	3: (* === Wait & process MB response *)
		IF NOT MB_Start THEN
			IF MB_MASTER.MB_Error=0 THEN
				CASE VARS[VarCnt].FunCode OF
					1,2,3,4:
						IF VARS[VarCnt].Variable_Size=200 THEN
							COPY_32SWAP16(ADR(MB_Resp.Data), VARS[VarCnt].Variable);
						ELSIF VARS[VarCnt].Variable_Size>1 THEN
							MEMCPY(ADR(MB_Resp.Data), VARS[VarCnt].Variable, 2*VARS[VarCnt].Variable_Size);
						ELSE
							VARS[VarCnt].Variable^:=MB_Resp.Data[0];
						END_IF
				END_CASE
				MB_Lock:=FALSE;
				(* Signal error recovery *)
				IF VARS_Alarm=TRUE AND VarCnt=VarAlarm THEN
					LogEv(EL_Wrn,EO_MODBUS,ID,5,'');
					VARS_Alarm:=FALSE;
				END_IF
				(* Next var *)
				VarCnt:=VarCnt+1;
				VarSta:=2;
			ELSE
				IF VarRetry<3 THEN
					VarRetry:=VarRetry+1;
					MB_Start:=TRUE;
				ELSE
					MB_Lock:=FALSE;
					(* Signal error *)
					IF VARS_Alarm=FALSE THEN
						LogEv(EL_Wrn,EO_MODBUS,ID,3,INT_TO_STRING(MB_MASTER.MB_Error));
						VARS_Alarm:=TRUE;
						VarAlarm:=VarCnt-1;
					END_IF
					(* Next var *)
					VarCnt:=VarCnt+1;
					VarSta:=2;
				END_IF
			END_IF
		END_IF

ELSE
	VarSta:=0;
END_CASE*)
;
END_ACTION

(* POU Plant_Objects/obj_MODBUS_TCP, ST *)
FUNCTION_BLOCK obj_MODBUS_TCP
(* === MODBUS-TCP PROTOCOL INTERFACE ===
   v1.0[10/06/15] - Create
*)
VAR CONSTANT
	VARS_Max	: BYTE := 32;
END_VAR
VAR_INPUT
	(* Settings *)
	ID			: BYTE;
	IP			: STRING;
	PORT		: WORD:=502;
	(* Interface *)
	MB_MASTER	: ETHERNET_MODBUSMASTER_TCP;
	MB_READBUF	: ARRAY [0..128] OF WORD;
	MB_WRITEBUF : ARRAY [0..128] OF WORD;
	MB_Start	: BOOL;
	MB_Lock		: BOOL;
	(* Variables management *)
	VARS_En		: BOOL;
	VARS		: ARRAY [0..VARS_Max] OF typ_MODBUS_VAR;
	VARS_Check	: BOOL;
	VARS_Alarm	: BOOL;
	(* Variables allocation *)
	VAR_Pointer : POINTER TO ARRAY[0..99] OF WORD;
	VAR_Cfg		: POINTER TO typ_MODBUS_VAR;
END_VAR
VAR_OUTPUT
	(* Status *)
	Status_Log	: BYTE;
	Status_Vis	: DWORD;
END_VAR
VAR
	sta         : BYTE :=0;
	i			: BYTE;
	j			: BYTE;
	Alarm		: FLT_EVENT;

	VarTmr		: TON := (PT:=T#1s);
	VarSta		: BYTE; (* Status *)
	VarCnt		: BYTE; (* Scan counter *)
	VarRetry	: BYTE;
	VarAlarm	: BYTE; (* Last variable with errors *)
END_VAR
MB_MASTER( strIP_ADDRESS:=IP, wPORT:=PORT, tTIME_OUT:=T#1s, (*xCONNECT:=TRUE,*)
		   ptREAD_DATA:=ADR(MB_READBUF), ptSEND_DATA:=ADR(MB_WRITEBUF), xSEND:=MB_Start );

IF sta=0 THEN
	MB_MASTER.xCONNECT:=TRUE;
	sta:=1;
END_IF

(* Process variable management *)
IF VARS_En THEN VARS_Process(); END_IF

(* Check status *)
Alarm(IN:=(MB_MASTER.wERROR<>0));
IF Alarm.EVH THEN
	(*LogEv(SEL(MB_MASTER.wERROR>0,EL_Wrn,EL_Alarm),EO_MODBUS_TCP,ID,1,WORD_TO_STRING(MB_MASTER.wERROR));*)
	(*LogEv(EL_Alarm,EO_MODBUS_TCP,ID,1,WORD_TO_STRING(MB_MASTER.wERROR));*);
END_IF
IF Alarm.EVL THEN
	(*LogEv(EL_Log,EO_MODBUS_TCP,ID,2,'');*);
END_IF

(* Log/visu status *)
   IF Alarm.IN   THEN Status_Log:=2; Status_Vis:=COLOR_RED;
ELSIF Vars_Alarm THEN Status_Log:=1; Status_Vis:=COLOR_YELLOW;
  				 ELSE Status_Log:=0; Status_Vis:=COLOR_GREEN;
END_IF
END_FUNCTION_BLOCK
ACTION VAR_Search:
(* Search VAR with specific pointer if not found return first free VAR
	[Last VAR is not active... used as safe area...] 
*)
j:=VARS_Max;
FOR i := 0 TO VARS_Max-1 DO
	IF VARS[i].Variable=0 AND j>i THEN j:=i; END_IF
	IF VARS[i].Variable=VAR_Pointer THEN
		VAR_Cfg:=ADR(VARS[i]);
		RETURN;
	END_IF
END_FOR
VAR_Cfg:=ADR(VARS[j]);
END_ACTION
ACTION VARS_Process:
(* Update var timers *)
(*VarTmr(IN:=(NOT VarTmr.Q));
IF VarTmr.Q THEN
	FOR i := 0 TO VARS_Max DO
		IF VARS[i].Refresh_Cnt>0 THEN VARS[i].Refresh_Cnt:=VARS[i].Refresh_Cnt-1; END_IF
	END_FOR
	VARS_Check:=TRUE;
END_IF


(* Process status *)
CASE VarSta OF
	0: (* === Init *)
		VarCnt:=0;
		VarSta:=1;

	1: (* === Wait check signal *)
		IF VARS_Check THEN
			VARS_Check:=FALSE;
			VarCnt:=0;
			VarSta:=2;
		END_IF

	2: (* === Check loop *)
		IF NOT (MB_Lock OR MB_Start) THEN
			WHILE VarCnt<=(VARS_Max-1) AND VarSta=2 DO
				(* Check only active vars *)
				IF VARS[VarCnt].Variable<>0 THEN
					(* Check var auto-refresh on timer checks *)
					IF VARS[VarCnt].Refresh_Time>0 AND VARS[VarCnt].Refresh_Cnt=0 THEN
						VARS[VarCnt].Refresh_Cnt:=VARS[VarCnt].Refresh_Time;
						VarSta:=3;
					END_IF
					(* Check refresh for change or request *)
					CASE VARS[VarCnt].FunCode OF
						5,6,15,16: (* Write functions *)
							IF VARS[VarCnt].Variable_Size=1 THEN
								IF VARS[VarCnt].Variable^<>VARS[VarCnt].Variable_Mirror THEN
									VARS[VarCnt].Variable_Mirror:=VARS[VarCnt].Variable^;
									VarSta:=3;
								END_IF
							ELSE
								IF VARS[VarCnt].Variable_Mirror<>0 THEN
									VARS[VarCnt].Variable_Mirror:=0;
									VarSta:=3;
								END_IF
							END_IF
						1,2,3,4: (* Write functions *)
							IF VARS[VarCnt].Variable_Mirror<>0 THEN
								VARS[VarCnt].Variable_Mirror:=0;
								VarSta:=3;
							END_IF
					END_CASE
				END_IF
				(* Process query *)
				IF VarSta=3 THEN
					MB_Lock:=TRUE;
					MB_MASTER.bUNIT_ID:=VARS[VarCnt].SlaveAddress;
					MB_MASTER.bFUNCTION_CODE:=VARS[VarCnt].FunCode;
					CASE VARS[VarCnt].FunCode OF
						16#5,16#6,16#F,16#10:
							MB_MASTER.wREAD_ADDRESS:=0;
							MB_MASTER.wREAD_QUANTITY:=0;
							MB_MASTER.wWRITE_ADDRESS:=VARS[VarCnt].FunAddress;
							MB_MASTER.wWRITE_QUANTITY:=VARS[VarCnt].Variable_Size;
							IF VARS[VarCnt].Variable_Size=200 THEN
								COPY_32SWAP16(VARS[VarCnt].Variable, ADR(MB_WRITEBUF));
							ELSIF VARS[VarCnt].Variable_Size>1 THEN
								MEMCPY(VARS[VarCnt].Variable, ADR(MB_WRITEBUF), 2*VARS[VarCnt].Variable_Size);
							ELSE
								MB_WRITEBUF[0]:=VARS[VarCnt].Variable^;
							END_IF
						16#1,16#2,16#3,16#4:
							MB_MASTER.wREAD_ADDRESS:=VARS[VarCnt].FunAddress;
							IF VARS[VarCnt].Variable_Size=200 THEN MB_MASTER.wREAD_QUANTITY:=2; ELSE
							  MB_MASTER.wREAD_QUANTITY:=VARS[VarCnt].Variable_Size;
							END_IF
							MB_MASTER.wWRITE_ADDRESS:=0;
							MB_MASTER.wWRITE_QUANTITY:=0;
					END_CASE
					VarRetry:=0;
					MB_Start:=TRUE;
				ELSE
					VarCnt:=VarCnt+1;
				END_IF
			END_WHILE
			(* Check loop completed -> no actions *)
			IF VarSta=2 THEN VarSta:=1; END_IF
		END_IF

	3: (* === Wait & process MB response *)
		IF NOT MB_Start THEN
			IF MB_MASTER.wERROR=0 THEN
				CASE VARS[VarCnt].FunCode OF
					1,2,3,4:
						IF VARS[VarCnt].Variable_Size=200 THEN
							COPY_32SWAP16(ADR(MB_READBUF), VARS[VarCnt].Variable);
						ELSIF VARS[VarCnt].Variable_Size>1 THEN
							MEMCPY(ADR(MB_READBUF), VARS[VarCnt].Variable, 2*VARS[VarCnt].Variable_Size);
						ELSE
							VARS[VarCnt].Variable^:=MB_READBUF[0];
						END_IF
				END_CASE
				MB_Lock:=FALSE;
				(* Signal error recovery *)
				IF VARS_Alarm=TRUE AND VarCnt=VarAlarm THEN
					LogEv(EL_Wrn,EO_MODBUS_TCP,ID,5,'');
					VARS_Alarm:=FALSE;
				END_IF
				(* Next var *)
				VarCnt:=VarCnt+1;
				VarSta:=2;
			ELSE
				IF VarRetry<10 THEN
					VarRetry:=VarRetry+1;
					MB_Start:=TRUE;
				ELSE
					MB_Lock:=FALSE;
					(* Signal error *)
					IF VARS_Alarm=FALSE THEN
						LogEv(EL_Wrn,EO_MODBUS_TCP,ID,3,WORD_TO_STRING(MB_MASTER.wERROR));
						VARS_Alarm:=TRUE;
						VarAlarm:=VarCnt-1;
					END_IF
					(* Next var *)
					VarCnt:=VarCnt+1;
					VarSta:=2;
				END_IF
			END_IF
		END_IF

ELSE
	VarSta:=0;
END_CASE*)	;
END_ACTION

(* POU Plant_Objects/obj_PLC_ELVI, ST *)
FUNCTION_BLOCK obj_PLC_ELVI
VAR CONSTANT
	WAIT_STATE		:	BYTE := 0;
	FIRST_WRITE		:	BYTE := 1;
	SECOND_WRITE	:	BYTE := 2;
	FIRST_READ		:	BYTE := 3;
	SECOND_READ		:	BYTE := 4;
	END_READ		:	BYTE := 5;

	READ_STATUS		:	BYTE := 10;
	READ_INFO		:	BYTE := 11;
	READ_MAINS		:	BYTE := 12;
	READ_GW_BATT	:	BYTE := 13;
	READ_GW_BATT_2	:	BYTE := 14;
	READ_PCS		:	BYTE := 15;

	ERROR_STATE	:	BYTE := 100;
END_VAR
VAR_INPUT
	ID			:	BYTE;
	Address		:	BYTE;

	Refresh_Now		:	BOOL;
	Refresh_Period	:	TIME := T#1s;
END_VAR
VAR_IN_OUT
	ModBus		:	obj_MODBUS_TCP;
END_VAR
VAR_OUTPUT
	Status_Log	:	WORD;
	Status_Vis	:	DWORD;

	NodeConnected	:	BOOL;
END_VAR
VAR
	state			:	BYTE;
	Timer			:	TON := (PT:=T#1s);
	retry 			:	BYTE;

	ResetCounter 	:	WORD := 5000;
	Status			:	BOOL;			(* 0:Normal working, 1:Autoreset routine	*)
	fSystemStatus	:	FLT_EVENT;
	WaitTime		:	TON := (PT:=T#3m);

	WriteBuf		:	ARRAY [0..19] OF WORD;
	Temp			:	DWORD;

END_VAR
(* ModBus state machine	*)
Stm1();

(* Check if a auto reset needed or reset request	*)
Reset();

IF Status_Log = 2 THEN Status_Vis := COLOR_RED;
ELSIF Status_Log = 1 THEN Status_Vis := COLOR_YELLOW;
ELSE Status_Vis := COLOR_GREEN;
END_IF
END_FUNCTION_BLOCK
ACTION Reset:
fSystemStatus(IN:=(Sistem_Status=7));

(* An error has occured	-->> Start AutoReset routine*)
IF fSystemStatus.EVH THEN

	IF NOT Status THEN
		(* If not returned to error state after autoreset routine	*)

		wbResetAlarm := TRUE;			(* Set flag high -->> Reset device	*)
		Status := TRUE;					(* Keep memory of the fact an autoreset routine is currently running	*)
	
		WaitTime(IN:=TRUE);				(* Start delay time before checking another time system status	*)
	END_IF
END_IF

(* Count time to keep high "wbResetAlarm" variable	*)
IF wbResetAlarm = TRUE THEN
	ResetCounter := ResetCounter - 1;

	IF ResetCounter = 0 THEN
		ResetCounter := 5000;
		wbResetAlarm := FALSE;		(* Clear "ResetAlarm" command after have sent it to the slave *)
	END_IF
END_IF


IF Status AND WaitTime.Q THEN
	(* 3 minutes are elapsed	*)
	WaitTime(IN:=FALSE);		(* Stop timer	*)

	IF Sistem_Status = 7 THEN ;
	ELSE ;
	END_IF

	Status := FALSE;			(* Autoreset routine ended	*)
END_IF
END_ACTION
ACTION Stm:
CASE state OF

	WAIT_STATE:	(* Wait State	*)
		Timer(IN:=NOT (Timer.Q OR Refresh_Now));

		IF Timer.Q OR Refresh_Now THEN

			(* Refresh timer and variable	*)
			Timer.PT:=Refresh_Period;
			Refresh_Now:=FALSE;

			(* Toggle communication bit	*)
			wbToggle_Bit_Comunication_SCADA:= NOT wbToggle_Bit_Comunication_SCADA;

			(* Prepare write buffer with data have to be sent	*)
			WriteBuf[0] := Da16Bit_A_Word(		wbToggle_Bit_Comunication_SCADA, (*bit_00*)
												wbStart_StopSystem,
												wbResetAlarm,
												0,
												0,
												0,
												wbRequestBatteryStayinVmode,
												wbRequestEOCBattery,
												wbRequestResetMoxa,
												0,
												0,
												0,
												0,
												0,
												0,
												0	);

			WriteBuf[1] := WORD_OF_DWORD(ConversioneReal_DWord(Ref_AvctivePower),0);
			WriteBuf[2] := WORD_OF_DWORD(ConversioneReal_DWord(Ref_AvctivePower),1);

			state := FIRST_WRITE;
		END_IF

	FIRST_WRITE:	(* Write update parameters to Elvi PLC and toggle communication variable	*)
		IF NOT (ModBus.MB_Lock OR ModBus.MB_Start) THEN
			ModBus.MB_Lock:=TRUE;

			ModBus.ID:=ID;
			ModBus.MB_MASTER.bUNIT_ID := Address;
			ModBus.MB_MASTER.bFUNCTION_CODE:=16#10;
			ModBus.MB_MASTER.wWRITE_ADDRESS:=16#0;
			ModBus.MB_MASTER.wWRITE_QUANTITY:=1;
			ModBus.MB_WRITEBUF[0] := WriteBuf[0];

			ModBus.MB_Start:=TRUE;

			state := SECOND_WRITE;
		END_IF

	SECOND_WRITE:
		IF NOT ModBus.MB_Start THEN
			IF ModBus.MB_MASTER.wERROR<>MB_NO_ERROR THEN
				state := ERROR_STATE;
			ELSE
				NodeConnected := ModBus.MB_MASTER.xIS_CONNECTED;

				ModBus.MB_MASTER.bUNIT_ID := Address;
				ModBus.MB_MASTER.bFUNCTION_CODE:=16#10;
				ModBus.MB_MASTER.wWRITE_ADDRESS:=10;
				ModBus.MB_MASTER.wWRITE_QUANTITY:=2;
				ModBus.MB_WRITEBUF[0] := WriteBuf[1];
				ModBus.MB_WRITEBUF[1] := WriteBuf[2];

				ModBus.MB_Start:=TRUE;

				state := READ_STATUS;

			END_IF
		END_IF

	READ_STATUS:
		IF NOT ModBus.MB_Start THEN
			IF ModBus.MB_MASTER.wERROR<>MB_NO_ERROR THEN
				state := ERROR_STATE;
			ELSE
				NodeConnected := ModBus.MB_MASTER.xIS_CONNECTED;

				ModBus.MB_MASTER.bUNIT_ID := Address;
				ModBus.MB_MASTER.bFUNCTION_CODE:=16#3;
				ModBus.MB_MASTER.wREAD_ADDRESS:=399;
				ModBus.MB_MASTER.wREAD_QUANTITY:=121;
				ModBus.MB_Start:=TRUE;

				state := SECOND_READ;
			END_IF
		END_IF

	(*SECOND_READ:
		IF NOT ModBus.MB_Start THEN
			IF ModBus.MB_MASTER.wERROR<>MB_NO_ERROR THEN
				state := ERROR_STATE;
			ELSE
				NodeConnected := ModBus.MB_MASTER.xIS_CONNECTED;
*)
	SECOND_READ:
		IF NOT ModBus.MB_Start THEN
			IF ModBus.MB_MASTER.wERROR<>MB_NO_ERROR THEN
				state := ERROR_STATE;
			ELSE
				NodeConnected := ModBus.MB_MASTER.xIS_CONNECTED;

				(* Read data from Elvi PLC through TCP Modbus	*)
				(* PLC *)
				Sistem_Status		 	:= ModBus.MB_READBUF[1];
				BATTERY_STATUS 			:= ModBus.MB_READBUF[2];
				SYSTEM_STATUS_COMMAND 	:= ModBus.MB_READBUF[11];
				STATUS_DIGITAL_INPUT_1 	:= ModBus.MB_READBUF[16];
				STATUS_DIGITAL_OUTPUT_1 := ModBus.MB_READBUF[21];
				STATUS_SYSTEM_WARNNG_1 	:= ModBus.MB_READBUF[26];
				STATUS_SYSTEM_ALARM_1  	:= ModBus.MB_READBUF[31];
				STATUS_SYSTEM_ALARM_2  	:= ModBus.MB_READBUF[32];
				
				PM1_Voltage_L12			:= ConversioneDword_Real(BUILD_16TO32LE(ADR(ModBus.MB_READBUF[37])));
				PM1_Voltage_L23			:= ConversioneDword_Real(BUILD_16TO32LE(ADR(ModBus.MB_READBUF[39])));
				PM1_Voltage_L31			:= ConversioneDword_Real(BUILD_16TO32LE(ADR(ModBus.MB_READBUF[41])));
				PM1_Current_L12			:= ConversioneDword_Real(BUILD_16TO32LE(ADR(ModBus.MB_READBUF[43])));
				PM1_Current_L23			:= ConversioneDword_Real(BUILD_16TO32(ADR(ModBus.MB_READBUF[45])));
				PM1_Current_L31			:= ConversioneDword_Real(BUILD_16TO32(ADR(ModBus.MB_READBUF[47])));
				PM1_Active_Power_Total	:= ConversioneDword_Real(ModBus.MB_READBUF[49]*65535+ModBus.MB_READBUF[50]);
				PM1_Reactive_Power_Total:= ConversioneDword_Real(ModBus.MB_READBUF[51]*65535+ModBus.MB_READBUF[52]);
				PM1_Apparent_Power_Total:= ConversioneDword_Real(ModBus.MB_READBUF[53]*65535+ModBus.MB_READBUF[54]);
				PM1_Frequency			:= ConversioneDword_Real(ModBus.MB_READBUF[55]*65535+ModBus.MB_READBUF[56]);
				PM1_Power_Factor_Total	:= ConversioneDword_Real(ModBus.MB_READBUF[57]*65535+ModBus.MB_READBUF[58]);
				
				(* GATEWAY BATTERY*)
				GW_Actual_DC_Voltage	:= ConversioneDword_Real(ModBus.MB_READBUF[71]*65535+ModBus.MB_READBUF[72]);
				GW_Actual_DC_Current	:= ConversioneDword_Real(ModBus.MB_READBUF[73]*65535+ModBus.MB_READBUF[74]);
				GW_Actual_Battery_SOC	:= ConversioneDword_Real(ModBus.MB_READBUF[75]*65535+ModBus.MB_READBUF[76]);
				GW_Actual_Heaters_Current:=ConversioneDword_Real(ModBus.MB_READBUF[77]*65535+ModBus.MB_READBUF[78]);
				GW_Vdc_Link_Request		:= ConversioneDword_Real(ModBus.MB_READBUF[79]*65535+ModBus.MB_READBUF[80]);
				GW_Limit_Discharge_Current:=ConversioneDword_Real(ModBus.MB_READBUF[81]*65535+ModBus.MB_READBUF[82]);
				GW_Limit_Charge_Current	:= ConversioneDword_Real(ModBus.MB_READBUF[83]*65535+ModBus.MB_READBUF[84]);
				GW_Min_DC_Voltage		:= ConversioneDword_Real(ModBus.MB_READBUF[85]*65535+ModBus.MB_READBUF[86]);
				GW_Max_DC_Voltage		:= ConversioneDword_Real(ModBus.MB_READBUF[87]*65535+ModBus.MB_READBUF[88]);
				GW_Actual_Battery_Capacity:=ConversioneDword_Real(ModBus.MB_READBUF[89]*65535+ModBus.MB_READBUF[90]);
				GW_Max_Battery_Voltage	:= ConversioneDword_Real(ModBus.MB_READBUF[93]*65535+ModBus.MB_READBUF[94]);
				GW_Min_Battery_Voltage	:= ConversioneDword_Real(ModBus.MB_READBUF[95]*65535+ModBus.MB_READBUF[96]);
				GW_Max_Battery_Temperature:=ConversioneDword_Real(ModBus.MB_READBUF[97]*65535+ModBus.MB_READBUF[98]);
				GW_Min_Battery_Temperature:=ConversioneDword_Real(ModBus.MB_READBUF[99]*65535+ModBus.MB_READBUF[100]);
				GW_Actual_DC_Power		:= ConversioneDword_Real(ModBus.MB_READBUF[101]*65535+ModBus.MB_READBUF[102]);
				
				GW_HOURSOp_Time 		:= ModBus.MB_READBUF[110];
				GW_MINOp_Time  			:= ModBus.MB_READBUF[111];
				GW_Status_Warning_1  	:= ModBus.MB_READBUF[112];
				GW_Status_Warning_2  	:= ModBus.MB_READBUF[113];
				GW_Status_Alarm_1 		:= ModBus.MB_READBUF[114];
				GW_Status_Alarm_2 		:= ModBus.MB_READBUF[115];
				GW_Status_Warning_A  	:= ModBus.MB_READBUF[116];
				GW_Status_Warning_B  	:= ModBus.MB_READBUF[117];
				GW_Status_Alarm_A 	 	:= ModBus.MB_READBUF[118];
				GW_CONTROLWORD  		:= ModBus.MB_READBUF[120];
				GW_STATUSWORD 			:= ModBus.MB_READBUF[121];

				ModBus.MB_MASTER.bUNIT_ID := Address;
				ModBus.MB_MASTER.bFUNCTION_CODE:=16#3;
				ModBus.MB_MASTER.wWRITE_ADDRESS:=598;
				ModBus.MB_MASTER.wWRITE_QUANTITY:=42;
				ModBus.MB_Start:=TRUE;

				state := END_READ;

			END_IF
		END_IF

	END_READ:
		IF NOT ModBus.MB_Start THEN
			IF ModBus.MB_MASTER.wERROR<>MB_NO_ERROR THEN
				state := ERROR_STATE;
			ELSE
				(* PCS HPP 35*)
				PCS_Actual_Current_R	:= ConversioneDword_Real(ModBus.MB_READBUF[3]*65535+ModBus.MB_READBUF[2]);
				PCS_Actual_Current_S	:= ConversioneDword_Real(ModBus.MB_READBUF[5]*65535+ModBus.MB_READBUF[4]);
				PCS_Actual_Current_T	:= ConversioneDword_Real(ModBus.MB_READBUF[7]*65535+ModBus.MB_READBUF[6]);
				PCS_Actual_Voltage_RS	:= ConversioneDword_Real(ModBus.MB_READBUF[9]*65535+ModBus.MB_READBUF[8]);
				PCS_Actual_Voltage_ST	:= ConversioneDword_Real(ModBus.MB_READBUF[11]*65535+ModBus.MB_READBUF[10]);
				PCS_Actual_Voltage_TR	:= ConversioneDword_Real(ModBus.MB_READBUF[13]*65535+ModBus.MB_READBUF[12]);
				PCS_Frequency			:= ConversioneDword_Real(ModBus.MB_READBUF[15]*65535+ModBus.MB_READBUF[14]);
				PCS_P_Actual			:= ConversioneDword_Real(ModBus.MB_READBUF[17]*65535+ModBus.MB_READBUF[16]);
				PCS_Q_Actual			:= ConversioneDword_Real(ModBus.MB_READBUF[19]*65535+ModBus.MB_READBUF[18]);
				PCS_A_Actual			:= ConversioneDword_Real(ModBus.MB_READBUF[21]*65535+ModBus.MB_READBUF[20]);
				PCS_Battery_Voltage		:= ConversioneDword_Real(ModBus.MB_READBUF[23]*65535+ModBus.MB_READBUF[22]);
				PCS_Battery_Current		:= ConversioneDword_Real(ModBus.MB_READBUF[25]*65535+ModBus.MB_READBUF[24]);
				PCS_Battery_Power		:= ConversioneDword_Real(ModBus.MB_READBUF[27]*65535+ModBus.MB_READBUF[26]);
				PCS_PV_Voltage			:= ConversioneDword_Real(ModBus.MB_READBUF[29]*65535+ModBus.MB_READBUF[28]);
				PCS_PV_Current			:= ConversioneDword_Real(ModBus.MB_READBUF[31]*65535+ModBus.MB_READBUF[30]);
				PCS_PV_Power			:= ConversioneDword_Real(ModBus.MB_READBUF[33]*65535+ModBus.MB_READBUF[32]);
				PCS_HPP_Status 			:= ModBus.MB_READBUF[34];
				PCS_Drive_Status  		:= ModBus.MB_READBUF[35];
				PCS_Chopper_Status 		:= ModBus.MB_READBUF[36];
				PCS_Run_Mode 	 		:= ModBus.MB_READBUF[37];
				PCS_Drive_Warning_1  	:= ModBus.MB_READBUF[38];
				PCS_Drive_Alarm_1 		:= ModBus.MB_READBUF[39];
				PCS_HPP_Warning_1   	:= ModBus.MB_READBUF[40];
				PCS_HPP_Alarm_1  		:= ModBus.MB_READBUF[41];

				retry := 0;
				ModBus.MB_Lock := FALSE;
				state := WAIT_STATE;

			END_IF
		END_IF

	ERROR_STATE:

		ModBus.MB_Lock:=FALSE;

			(* Retries *)
		retry:=retry+1;

		IF retry>3 THEN
			retry:=0;

			IF Status_Log<>2 THEN
				LogEv(EL_Alarm,100,ID,4,'Modbus_communication_error');
			END_IF

			Status_Log:=2;
		END_IF

		state := WAIT_STATE;


END_CASE
END_ACTION
ACTION Stm1:
CASE state OF

	WAIT_STATE:	(* Wait State	*)
		Timer(IN:=NOT (Timer.Q OR Refresh_Now));

		IF Timer.Q OR Refresh_Now THEN

			(* Refresh timer and variable	*)
			Timer.PT:=Refresh_Period;
			Refresh_Now:=FALSE;

			(* Toggle communication bit	*)
			wbToggle_Bit_Comunication_SCADA:= NOT wbToggle_Bit_Comunication_SCADA;

			(* Prepare write buffer with data have to be sent	*)
			WriteBuf[0] := Da16Bit_A_Word(		wbToggle_Bit_Comunication_SCADA, (*bit_00*)
												wbStart_StopSystem,
												wbResetAlarm,
												0,
												0,
												0,
												wbRequestBatteryStayinVmode,
												wbRequestEOCBattery,
												wbRequestResetMoxa,
												0,
												0,
												0,
												0,
												0,
												0,
												0	);

			WriteBuf[1] := WORD_OF_DWORD(ConversioneReal_DWord(Ref_AvctivePower),0);
			WriteBuf[2] := WORD_OF_DWORD(ConversioneReal_DWord(Ref_AvctivePower),1);

			state := FIRST_WRITE;
		END_IF

	FIRST_WRITE:	(* Write update parameters to Elvi PLC and toggle communication variable	*)
		IF NOT (ModBus.MB_Lock OR ModBus.MB_Start) THEN
			ModBus.MB_Lock:=TRUE;

			ModBus.ID:=ID;
			ModBus.MB_MASTER.bUNIT_ID := Address;
			ModBus.MB_MASTER.bFUNCTION_CODE:=16#10;
			ModBus.MB_MASTER.wWRITE_ADDRESS:=16#0;
			ModBus.MB_MASTER.wWRITE_QUANTITY:=1;
			ModBus.MB_WRITEBUF[0] := WriteBuf[0];

			ModBus.MB_Start:=TRUE;

			state := SECOND_WRITE;
		END_IF

	SECOND_WRITE:
		IF NOT ModBus.MB_Start THEN
			IF ModBus.MB_MASTER.wERROR<>MB_NO_ERROR THEN
				state := ERROR_STATE;
			ELSE
				NodeConnected := ModBus.MB_MASTER.xIS_CONNECTED;

				ModBus.MB_MASTER.bUNIT_ID := Address;
				ModBus.MB_MASTER.bFUNCTION_CODE:=16#10;
				ModBus.MB_MASTER.wWRITE_ADDRESS:=10;
				ModBus.MB_MASTER.wWRITE_QUANTITY:=2;
				ModBus.MB_WRITEBUF[0] := WriteBuf[1];
				ModBus.MB_WRITEBUF[1] := WriteBuf[2];

				ModBus.MB_Start:=TRUE;

				state := READ_STATUS;

			END_IF
		END_IF

	READ_STATUS:
		IF NOT ModBus.MB_Start THEN
			IF ModBus.MB_MASTER.wERROR<>MB_NO_ERROR THEN
				state := ERROR_STATE;
			ELSE
				NodeConnected := ModBus.MB_MASTER.xIS_CONNECTED;

				ModBus.MB_MASTER.bUNIT_ID := Address;
				ModBus.MB_MASTER.bFUNCTION_CODE:=16#3;
				ModBus.MB_MASTER.wREAD_ADDRESS:=399;
				ModBus.MB_MASTER.wREAD_QUANTITY:=2;
				ModBus.MB_Start:=TRUE;

				state := READ_INFO;
			END_IF
		END_IF

	READ_INFO:
		IF NOT ModBus.MB_Start THEN
			IF ModBus.MB_MASTER.wERROR<>MB_NO_ERROR THEN
				state := ERROR_STATE;
			ELSE
				(* Read data from Elvi PLC through TCP Modbus	*)
				(* PLC *)
				Sistem_Status		 	:= ModBus.MB_READBUF[0];
				BATTERY_STATUS 			:= ModBus.MB_READBUF[1];

				ModBus.MB_MASTER.bUNIT_ID := Address;
				ModBus.MB_MASTER.bFUNCTION_CODE:=16#3;
				ModBus.MB_MASTER.wREAD_ADDRESS:=409;
				ModBus.MB_MASTER.wREAD_QUANTITY:=22;
				ModBus.MB_Start:=TRUE;

				state := READ_MAINS;

			END_IF
		END_IF

	READ_MAINS:
		IF NOT ModBus.MB_Start THEN
			IF ModBus.MB_MASTER.wERROR<>MB_NO_ERROR THEN
				state := ERROR_STATE;
			ELSE
				SYSTEM_STATUS_COMMAND 	:=ModBus.MB_READBUF[0];
				STATUS_DIGITAL_INPUT_1 	:=ModBus.MB_READBUF[5];
				STATUS_DIGITAL_OUTPUT_1 :=ModBus.MB_READBUF[10];
				STATUS_SYSTEM_WARNNG_1 	:=ModBus.MB_READBUF[15];
				STATUS_SYSTEM_ALARM_1  	:=ModBus.MB_READBUF[20];
				STATUS_SYSTEM_ALARM_2  	:=ModBus.MB_READBUF[21];

				ModBus.MB_MASTER.bUNIT_ID := Address;
				ModBus.MB_MASTER.bFUNCTION_CODE:=16#3;
				ModBus.MB_MASTER.wREAD_ADDRESS:=435;
				ModBus.MB_MASTER.wREAD_QUANTITY:=22;
				ModBus.MB_Start:=TRUE;

				state := READ_GW_BATT;

			END_IF
		END_IF

	READ_GW_BATT:
		IF NOT ModBus.MB_Start THEN
			IF ModBus.MB_MASTER.wERROR<>MB_NO_ERROR THEN
				state := ERROR_STATE;
			ELSE

				PM1_Voltage_L12			:= ConversioneDword_Real(BUILD_16TO32LE(ADR(ModBus.MB_READBUF[0])));
				PM1_Voltage_L23			:= ConversioneDword_Real(BUILD_16TO32LE(ADR(ModBus.MB_READBUF[2])));
				PM1_Voltage_L31			:= ConversioneDword_Real(BUILD_16TO32LE(ADR(ModBus.MB_READBUF[4])));
				PM1_Current_L12			:= ConversioneDword_Real(BUILD_16TO32LE(ADR(ModBus.MB_READBUF[6])));
				PM1_Current_L23			:= ConversioneDword_Real(BUILD_16TO32LE(ADR(ModBus.MB_READBUF[8])));
				PM1_Current_L31			:= ConversioneDword_Real(BUILD_16TO32LE(ADR(ModBus.MB_READBUF[10])));
				PM1_Active_Power_Total	:= ConversioneDword_Real(BUILD_16TO32LE(ADR(ModBus.MB_READBUF[12])));
				PM1_Reactive_Power_Total:= ConversioneDword_Real(BUILD_16TO32LE(ADR(ModBus.MB_READBUF[14])));
				PM1_Apparent_Power_Total:= ConversioneDword_Real(BUILD_16TO32LE(ADR(ModBus.MB_READBUF[16])));
				PM1_Frequency			:= ConversioneDword_Real(BUILD_16TO32LE(ADR(ModBus.MB_READBUF[18])));
				PM1_Power_Factor_Total	:= ConversioneDword_Real(BUILD_16TO32LE(ADR(ModBus.MB_READBUF[20])));

				ModBus.MB_MASTER.bUNIT_ID := Address;
				ModBus.MB_MASTER.bFUNCTION_CODE:=16#3;
				ModBus.MB_MASTER.wREAD_ADDRESS:=469;
				ModBus.MB_MASTER.wREAD_QUANTITY:=30;
				ModBus.MB_Start:=TRUE;

				state := READ_GW_BATT_2;
			END_IF
		END_IF

	READ_GW_BATT_2:
		IF NOT ModBus.MB_Start THEN
			IF ModBus.MB_MASTER.wERROR<>MB_NO_ERROR THEN
				state := ERROR_STATE;
			ELSE
				GW_Actual_DC_Voltage		:= ConversioneDword_Real(BUILD_16TO32LE(ADR(ModBus.MB_READBUF[0])));
				GW_Actual_DC_Current		:= ConversioneDword_Real(BUILD_16TO32LE(ADR(ModBus.MB_READBUF[2])));
				GW_Actual_Battery_SOC		:= ConversioneDword_Real(BUILD_16TO32LE(ADR(ModBus.MB_READBUF[4])));
				GW_Actual_Heaters_Current	:= ConversioneDword_Real(BUILD_16TO32LE(ADR(ModBus.MB_READBUF[6])));
				GW_Vdc_Link_Request			:= ConversioneDword_Real(BUILD_16TO32LE(ADR(ModBus.MB_READBUF[8])));
				GW_Limit_Discharge_Current	:= ConversioneDword_Real(BUILD_16TO32LE(ADR(ModBus.MB_READBUF[10])));
				GW_Limit_Charge_Current		:= ConversioneDword_Real(BUILD_16TO32LE(ADR(ModBus.MB_READBUF[12])));
				GW_Min_DC_Voltage			:= ConversioneDword_Real(BUILD_16TO32LE(ADR(ModBus.MB_READBUF[14])));
				GW_Max_DC_Voltage			:= ConversioneDword_Real(BUILD_16TO32LE(ADR(ModBus.MB_READBUF[16])));
				GW_Actual_Battery_Capacity	:= ConversioneDword_Real(BUILD_16TO32LE(ADR(ModBus.MB_READBUF[18])));
				GW_Max_Battery_Voltage		:= ConversioneDword_Real(BUILD_16TO32LE(ADR(ModBus.MB_READBUF[20])));
				GW_Min_Battery_Voltage		:= ConversioneDword_Real(BUILD_16TO32LE(ADR(ModBus.MB_READBUF[22])));
				GW_Max_Battery_Temperature	:= ConversioneDword_Real(BUILD_16TO32LE(ADR(ModBus.MB_READBUF[24])));
				GW_Min_Battery_Temperature	:= ConversioneDword_Real(BUILD_16TO32LE(ADR(ModBus.MB_READBUF[26])));
				GW_Actual_DC_Power			:= ConversioneDword_Real(BUILD_16TO32LE(ADR(ModBus.MB_READBUF[28])));

				ModBus.MB_MASTER.bUNIT_ID := Address;
				ModBus.MB_MASTER.bFUNCTION_CODE:=16#3;
				ModBus.MB_MASTER.wREAD_ADDRESS:=508;
				ModBus.MB_MASTER.wREAD_QUANTITY:=11;
				ModBus.MB_Start:=TRUE;

				state := READ_PCS;

			END_IF
		END_IF

	READ_PCS:
		IF NOT ModBus.MB_Start THEN
			IF ModBus.MB_MASTER.wERROR<>MB_NO_ERROR THEN
				state := ERROR_STATE;
			ELSE
				GW_HOURSOp_Time 		:= ModBus.MB_READBUF[0];
				GW_MINOp_Time  			:= ModBus.MB_READBUF[1];
				GW_Status_Warning_1  	:= ModBus.MB_READBUF[2];
				GW_Status_Warning_2  	:= ModBus.MB_READBUF[3];
				GW_Status_Alarm_1 		:= ModBus.MB_READBUF[4];
				GW_Status_Alarm_2 		:= ModBus.MB_READBUF[5];
				GW_Status_Warning_A  	:= ModBus.MB_READBUF[6];
				GW_Status_Warning_B  	:= ModBus.MB_READBUF[7];
				GW_Status_Alarm_A 	 	:= ModBus.MB_READBUF[8];
				GW_CONTROLWORD  		:= ModBus.MB_READBUF[10];
				GW_STATUSWORD 			:= ModBus.MB_READBUF[11];

				ModBus.MB_MASTER.bUNIT_ID := Address;
				ModBus.MB_MASTER.bFUNCTION_CODE:=16#3;
				ModBus.MB_MASTER.wWRITE_ADDRESS:=600;
				ModBus.MB_MASTER.wWRITE_QUANTITY:=41;
				ModBus.MB_Start:=TRUE;

				state := END_READ;

			END_IF
		END_IF

	END_READ:
		IF NOT ModBus.MB_Start THEN
			IF ModBus.MB_MASTER.wERROR<>MB_NO_ERROR THEN
				state := ERROR_STATE;
			ELSE
				(* PCS HPP 35*)
				PCS_Actual_Current_R	:= ConversioneDword_Real(BUILD_16TO32(ADR(ModBus.MB_READBUF[0])));
				PCS_Actual_Current_S	:= ConversioneDword_Real(BUILD_16TO32(ADR(ModBus.MB_READBUF[2])));
				PCS_Actual_Current_T	:= ConversioneDword_Real(BUILD_16TO32(ADR(ModBus.MB_READBUF[4])));
				PCS_Actual_Voltage_RS	:= ConversioneDword_Real(BUILD_16TO32(ADR(ModBus.MB_READBUF[6])));
				PCS_Actual_Voltage_ST	:= ConversioneDword_Real(BUILD_16TO32(ADR(ModBus.MB_READBUF[8])));
				PCS_Actual_Voltage_TR	:= ConversioneDword_Real(BUILD_16TO32(ADR(ModBus.MB_READBUF[10])));
				PCS_Frequency			:= ConversioneDword_Real(BUILD_16TO32(ADR(ModBus.MB_READBUF[12])));
				PCS_P_Actual			:= ConversioneDword_Real(BUILD_16TO32(ADR(ModBus.MB_READBUF[14])));
				PCS_Q_Actual			:= ConversioneDword_Real(BUILD_16TO32(ADR(ModBus.MB_READBUF[16])));
				PCS_A_Actual			:= ConversioneDword_Real(BUILD_16TO32(ADR(ModBus.MB_READBUF[18])));
				PCS_Battery_Voltage		:= ConversioneDword_Real(BUILD_16TO32(ADR(ModBus.MB_READBUF[20])));
				PCS_Battery_Current		:= ConversioneDword_Real(BUILD_16TO32(ADR(ModBus.MB_READBUF[22])));
				PCS_Battery_Power		:= ConversioneDword_Real(BUILD_16TO32(ADR(ModBus.MB_READBUF[24])));
				PCS_PV_Voltage			:= ConversioneDword_Real(BUILD_16TO32(ADR(ModBus.MB_READBUF[26])));
				PCS_PV_Current			:= ConversioneDword_Real(BUILD_16TO32(ADR(ModBus.MB_READBUF[28])));
				PCS_PV_Power			:= ConversioneDword_Real(BUILD_16TO32(ADR(ModBus.MB_READBUF[30])));
				PCS_HPP_Status 			:= ModBus.MB_READBUF[32];
				PCS_Drive_Status  		:= ModBus.MB_READBUF[33];
				PCS_Chopper_Status 		:= ModBus.MB_READBUF[34];
				PCS_Run_Mode 	 		:= ModBus.MB_READBUF[35];
				PCS_Drive_Warning_1  	:= ModBus.MB_READBUF[36];
				PCS_Drive_Alarm_1 		:= ModBus.MB_READBUF[37];
				PCS_HPP_Warning_1   	:= ModBus.MB_READBUF[38];
				PCS_HPP_Alarm_1  		:= ModBus.MB_READBUF[39];

				retry := 0;
				ModBus.MB_Lock := FALSE;
				state := WAIT_STATE;

			END_IF
		END_IF

	ERROR_STATE:

		ModBus.MB_Lock:=FALSE;

			(* Retries *)
		retry:=retry+1;

		IF retry>3 THEN
			retry:=0;

			IF Status_Log<>2 THEN
				LogEv(EL_Alarm,100,ID,4,'Modbus_communication_error');
			END_IF

			Status_Log:=2;
		END_IF

		state := WAIT_STATE;


END_CASE
END_ACTION

(* POU Plant_Objects/obj_ZTHL, ST *)
FUNCTION_BLOCK obj_ZTHL
(* === ZIGBEE AMBIENT SENSORS MT-200 ===
   v1.0[07/05/05] - Create
*)
VAR CONSTANT
	(* States *)
	WAIT_STATE			:	BYTE := 0;
	STATUS_REQUEST		:	BYTE := 1;
	LQI_REQUEST			:	BYTE := 2;
	MEAS_REQUEST		:	BYTE := 3;
	END_READ			:	BYTE := 4;
	ERROR_STATE			:	BYTE := 100;

	LQI_Threshold		:	WORD := 100;		(* Zigbee link quality minimum value *)
	LowBattVoltage		:	WORD := 270;		(* Battery is considered low when reaches 1.35V each *)
END_VAR
VAR_INPUT
	(* Settings *)
	ID				: BYTE;
	Address			: BYTE;

	Refresh_Period	: TIME:=t#5m;
	(* Controls *)
	Refresh_Auto	: BOOL:=TRUE; (* Enable automatic refresh *)
	Refresh_Now		: BOOL; 	  (* Force an immediate refresh *)

	(* Limits *)
	Tmin			: INT := 0;
	Tmax			: INT := 400;
END_VAR
VAR_IN_OUT
	(* Interface *)
	MODBUS			: obj_MODBUS_TCP;
END_VAR
VAR_OUTPUT
	OUT_TEMP		: INT;	(* Temperatura misurata [°C/10] *)
	OUT_HYGRO		: INT;	(* Umidità misurata [%] *)
	OUT_LUX			: INT;	(* Luce misurata [lux] *)
	OUT_VBATT		: INT;	(* Tensione misurata dalla batteria [V/100] *)

	OUT_LQI			: BYTE;

	NodeStatus		: WORD;
	fTemp			: BOOL;

	(* Status *)
	Status_Log		: BYTE;
	Status_Vis 		: DWORD;
END_VAR
VAR
	dly 	 		: TON := (PT:=t#5s);

	sta				: BYTE;
	retry	 		: BYTE;

	OldNodeStatus	: WORD;
	fLQI			: BOOL;
	fBatt			: BOOL;
	Quality			: FLT_EVENT;
	Battery			: FLT_EVENT;
	Temperature		: FLT_EVENT;
	Alarm			: FLT_EVENT;

	StatusOK		: BYTE;			(* 0: Status OK, >=1: Alarm and/or warning		Incremented by 1 when Alarm or Wrn occurs,
																					decremented by 1 when restored	*)
END_VAR
CASE sta OF
	WAIT_STATE: (* === Wait update signals *)
		dly(IN:=NOT (dly.Q OR Refresh_Now OR (NOT Refresh_Auto)));
		IF dly.Q OR Refresh_Now THEN
			dly.PT:=Refresh_Period;
			Refresh_Now:=FALSE;
			(*sta:=STATUS_REQUEST;*)
			sta:=LQI_REQUEST;
		END_IF

	STATUS_REQUEST:	(* Node status *)
		IF NOT (MODBUS.MB_Lock OR MODBUS.MB_Start) THEN
			MODBUS.MB_Lock:=TRUE;
			MODBUS.ID:=ID;
			MODBUS.MB_MASTER.bUNIT_ID := Address;
			MODBUS.MB_MASTER.bFUNCTION_CODE:=16#03;
			MODBUS.MB_MASTER.wREAD_ADDRESS:=16#0D;
			MODBUS.MB_MASTER.wREAD_QUANTITY:=16#1;
			MODBUS.MB_Start:=TRUE;
			sta:=LQI_REQUEST;
		END_IF

	LQI_REQUEST:	(* Link quality *)
		IF NOT MODBUS.MB_Start THEN
			IF MODBUS.MB_MASTER.wERROR<>MB_NO_ERROR THEN
				sta:=ERROR_STATE;
			ELSE
				(*NodeStatus	:=	MODBUS.MB_READBUF[0];*)

				MODBUS.ID:=ID;
				MODBUS.MB_MASTER.bUNIT_ID := Address;
				MODBUS.MB_MASTER.bFUNCTION_CODE:=16#03;
				MODBUS.MB_MASTER.wREAD_ADDRESS:=16#01;
				MODBUS.MB_MASTER.wREAD_QUANTITY:=16#1;
				MODBUS.MB_Start:=TRUE;

				sta:=MEAS_REQUEST;
			END_IF
		END_IF

	MEAS_REQUEST:	(* Measurements *)
		IF NOT MODBUS.MB_Start THEN
			IF MODBUS.MB_MASTER.wERROR<>MB_NO_ERROR THEN
				sta:=ERROR_STATE;
			ELSE

				OUT_LQI	:=	WORD_TO_BYTE(MODBUS.MB_READBUF[0]);

				MODBUS.ID:=ID;
				MODBUS.MB_MASTER.bUNIT_ID := Address;
				MODBUS.MB_MASTER.bFUNCTION_CODE:=16#03;
				MODBUS.MB_MASTER.wREAD_ADDRESS:=16#14;
				MODBUS.MB_MASTER.wREAD_QUANTITY:=16#5;
				MODBUS.MB_Start:=TRUE;

				sta:=END_READ;
			END_IF
		END_IF

	END_READ:	IF NOT MODBUS.MB_Start THEN
			IF MODBUS.MB_MASTER.wERROR<>MB_NO_ERROR THEN
				sta:=ERROR_STATE;
			ELSE
				OUT_TEMP	:=	WORD_TO_INT(MODBUS.MB_READBUF[0]);
				OUT_HYGRO	:=	WORD_TO_INT(MODBUS.MB_READBUF[1]);
				OUT_LUX		:=	WORD_TO_INT(MODBUS.MB_READBUF[2]);
				OUT_VBATT	:=	WORD_TO_INT(MODBUS.MB_READBUF[3]);
				sta:=WAIT_STATE;
				MODBUS.MB_Lock:=FALSE;
			END_IF
		END_IF

	ERROR_STATE:
			MODBUS.MB_Lock:=FALSE;
			(* Retries *)
			retry:=retry+1;
			IF retry>3 THEN
				retry:=0;
				IF Status_Log<>2 THEN
					LogEv(EL_Alarm,EO_ZTHL,ID,4,'');
				END_IF
				Status_Log:=2;
				Status_Vis:=COLOR_RED;
			END_IF
			sta:=WAIT_STATE;

ELSE
			sta:=WAIT_STATE;
END_CASE

(* Check Status *)
(*
IF NodeStatus <> OldNodeStatus THEN
	IF NodeStatus = 3 THEN
		LogEv(EL_Alarm,EO_ZTHL,ID,3,'');
		Status_Log:=2;
	ELSE
		Status_Log:=0;
	END_IF

	OldNodeStatus := NodeStatus;
END_IF*)

(* Check Link quality *)
IF OUT_LQI > LQI_Threshold THEN fLQI := TRUE;
ELSE fLQI := FALSE;
END_IF

Quality(IN:=fLQI);

IF Quality.EVL THEN
	LogEv(SEL(OUT_LQI<>0,EL_Alarm,EL_Wrn),EO_ZTHL,ID,SEL(OUT_LQI<>0,7,2),WORD_TO_STRING(OUT_LQI));
	Status_Log := SEL(OUT_LQI<>0,2,1);
	StatusOK := StatusOK + 1;
END_IF

IF Quality.EVH THEN StatusOK := SEL(StatusOK=0, StatusOK-1, 0); END_IF

(* If probe (node) is present proceed checking other warnings, otherwise don't transmit anything *)
IF OUT_LQI <> 0 THEN

	(* Check battery voltage *)
	IF OUT_VBATT < LowBattVoltage THEN fBatt := TRUE;
	ELSE fBatt := FALSE;
	END_IF
	
	Battery(IN:=fBatt);
	
	IF Battery.EVH THEN
		LogEv(EL_Wrn,EO_ZTHL,ID,6,'');
		StatusOK := StatusOK + 1;
	END_IF

	IF Battery.EVL THEN StatusOK := SEL(StatusOK=0, StatusOK-1, 0); END_IF

	(* Check Node temperature *)
	IF OUT_TEMP < Tmin OR OUT_TEMP > Tmax THEN
		fTemp := TRUE;
	ELSE
		fTemp := FALSE;
	END_IF

	Temperature(IN:=fTemp);

	IF Temperature.EVH THEN
		LogEv(EL_Wrn,EO_ZTHL,ID,5,INT_TO_STRING(OUT_TEMP));
		Status_Log := 1;
		StatusOK := StatusOK + 1;
	END_IF

	IF Temperature.EVL THEN StatusOK := SEL(StatusOK=0, StatusOK-1, 0); END_IF

END_IF

Alarm(IN:=(StatusOK=0));

IF Alarm.EVH THEN
	Status_Log := 0;
	LogEv(EL_Log,EO_ZTHL,ID,1,'');
END_IF

IF Status_Log = 2 THEN Status_Vis := COLOR_RED;
ELSIF Status_Log = 1 THEN Status_Vis := COLOR_YELLOW;
ELSE Status_Vis := COLOR_GREEN;
END_IF
END_FUNCTION_BLOCK
ACTION AddLogData:
Logger.s1:=INSERT('&ZTHL=',BYTE_TO_STRING(ID),4);
IF ID<10 THEN Logger.s1:=INSERT(Logger.s1,'0',4); END_IF

Logger.s1:=CONCAT(Logger.s1,BYTE_TO_STRING(OUT_LQI));			Logger.s1:=CONCAT(Logger.s1,';');
Logger.s1:=CONCAT(Logger.s1,INT_TO_STRING(OUT_TEMP ));			Logger.s1:=CONCAT(Logger.s1,';');
Logger.s1:=CONCAT(Logger.s1,INT_TO_STRING(OUT_HYGRO ));			Logger.s1:=CONCAT(Logger.s1,';');
Logger.s1:=CONCAT(Logger.s1,INT_TO_STRING(OUT_LUX));			Logger.s1:=CONCAT(Logger.s1,';');
Logger.s1:=CONCAT(Logger.s1,INT_TO_STRING(OUT_VBATT));			Logger.s1:=CONCAT(Logger.s1,';');

Logger.s1:=CONCAT(Logger.s1,BYTE_TO_STRING(Status_Log));
ADDSTRING(ADR(Logger.TData), ADR(Logger.s1), Logger.TLen);
END_ACTION

(* POU PLC_WDT, ST *)
FUNCTION PLC_WDT: DWORD VAR_INPUT dwEvent: DWORD; dwFilter: DWORD; dwOwner: DWORD; END_VAR
LogEv(EL_AlarmStop,EO_SYS,1,10,'Watchdog');
END_FUNCTION

(* POU Utils Functions/RAWTOHEX, ST *)
FUNCTION RAWTOHEX : WORD
VAR_INPUT
	pData: POINTER TO BYTE;
	DataLen: WORD;
	pString: POINTER TO BYTE;
END_VAR
VAR
	xl: WORD;
END_VAR
xl:=0;

WHILE DataLen>0 DO

	pString^ := (pData^ / 16#10) + 48 + (((pData^ / 16#10)/10)*7);
	pString:=pString+1;
	pString^ := (pData^ AND 16#0F)  + 48 + (((pData^ AND 16#0F)/10)*7);
	pString:=pString+1;
	pData:=pData+1;
	DataLen:=DataLen-1;
	xl:=xl+2;

END_WHILE

(*pString^:=0;*)

RAWTOHEX:=xl;
END_FUNCTION

(* POU Utils Functions/RAWTOHEXSTR, ST *)
FUNCTION RAWTOHEXSTR : STRING(128)
VAR_INPUT
	pData: POINTER TO BYTE;
	DataLen: BYTE;
END_VAR
VAR
	pt: POINTER TO BYTE;
	xl: BYTE;
END_VAR
pt:=ADR(RAWTOHEXSTR);

xl:=2;

WHILE DataLen>0 AND xl<128 DO

	pt^ := (pData^ / 16#10) + 48 + (((pData^ / 16#10)/10)*7);
	pt:=pt+1;
	pt^ := (pData^ AND 16#0F)  + 48 + (((pData^ AND 16#0F)/10)*7);
	pt:=pt+1;

	xl:=xl+2;

	DataLen:=DataLen-1;
	pData:=pData+1;

END_WHILE

pt^:=0;
END_FUNCTION

(* POU Utils/RTC_Update, ST *)
FUNCTION RTC_Update : BOOL
VAR
	T: DT;
	TS: STRING;
	TS2: STRING;
	Hour: BYTE;
	Minute: BYTE;
END_VAR
(* Get RTC time *)
T:=SysRtcGetTime(TRUE);
Sys.Time_CT_DT:=T;
(* Calculate variables *)
TS:=DT_TO_STRING(T);
Sys.Time_LogString:=DELETE(STR:=TS, LEN:=3, POS:=1);
TS2:=MID(STR:=TS, LEN:=4, POS:= 4); Sys.Time_Year 	:=STRING_TO_WORD(TS2);
TS2:=MID(STR:=TS, LEN:=2, POS:= 9); Sys.Time_Month	:=STRING_TO_BYTE(TS2);
TS2:=MID(STR:=TS, LEN:=2, POS:=12); Sys.Time_Day  	:=STRING_TO_BYTE(TS2);
Sys.Time_CT_Day:=(32*(Sys.Time_Month-1)+Sys.Time_Day-1);
TS2:=MID(STR:=TS, LEN:=2, POS:=15); Hour			:=STRING_TO_BYTE(TS2);
TS2:=MID(STR:=TS, LEN:=2, POS:=18); Minute		 	:=STRING_TO_BYTE(TS2);
Sys.Time_CT_Quarter:=Hour*4+(Minute/15);
END_FUNCTION

(* Visualisation IR_VISU
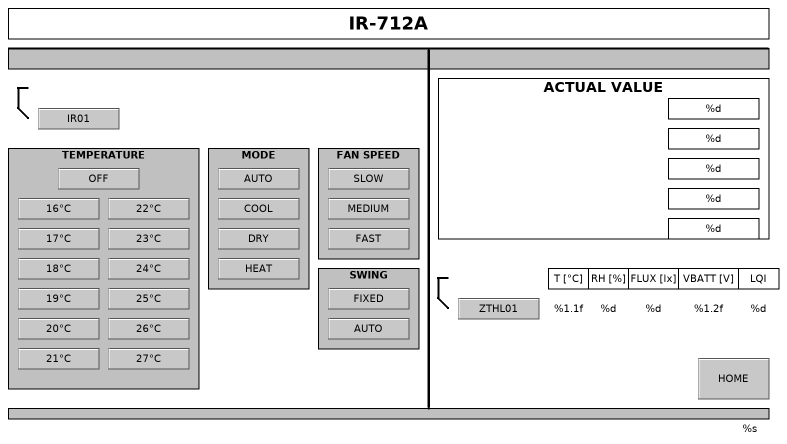
rectangle at (450,80)-(781,241): text "ACTUAL VALUE"
rounded rectangle at (20,150)-(211,391): text "TEMPERATURE"
rounded rectangle at (220,150)-(321,291): text "MODE"
rectangle at (530,420)-(771,441): text "%s"; shows Sys.Time_LogString
button at (50,110)-(131,131): text "IR01"
button at (70,170)-(151,191): text "OFF"; runs INTERN ASSIGN IR01.Off:=(TRUE)
button at (230,200)-(311,221): text "COOL"; runs INTERN ASSIGN IR01.Cmd_Mode:=(19)
button at (230,230)-(311,251): text "DRY"; runs INTERN ASSIGN IR01.Cmd_Mode:=(20)
button at (230,260)-(311,281): text "HEAT"; runs INTERN ASSIGN IR01.Cmd_Mode:=(21)
rounded rectangle at (330,150)-(431,261): text "FAN SPEED"
button at (340,170)-(421,191): text "SLOW"; runs INTERN ASSIGN IR01.Cmd_Fan:=(15)
button at (340,200)-(421,221): text "MEDIUM"; runs INTERN ASSIGN IR01.Cmd_Fan:=(16)
button at (340,230)-(421,251): text "FAST"; runs INTERN ASSIGN IR01.Cmd_Fan:=(17)
rectangle at (680,130)-(771,151): text "%d"; shows (IR01.SetCmdTemp)+13
button at (230,170)-(311,191): text "AUTO"; runs INTERN ASSIGN IR01.Cmd_Mode:=(18)
rounded rectangle at (330,270)-(431,351): text "SWING"
button at (340,290)-(421,311): text "FIXED"; runs INTERN ASSIGN IR01.Cmd_Swing:=(22)
button at (340,320)-(421,341): text "AUTO"; runs INTERN ASSIGN IR01.Cmd_Swing:=(23)
button at (30,200)-(111,221): text "16°C"; runs INTERN ASSIGN IR01.Cmd_Temp:=(3)
button at (30,230)-(111,251): text "17°C"; runs INTERN ASSIGN IR01.Cmd_Temp:=(4)
button at (30,260)-(111,281): text "18°C"; runs INTERN ASSIGN IR01.Cmd_Temp:=(5)
button at (30,290)-(111,311): text "19°C"; runs INTERN ASSIGN IR01.Cmd_Temp:=(6)
button at (30,320)-(111,341): text "20°C"; runs INTERN ASSIGN IR01.Cmd_Temp:=(7)
button at (30,350)-(111,371): text "21°C"; runs INTERN ASSIGN IR01.Cmd_Temp:=(8)
button at (120,200)-(201,221): text "22°C"; runs INTERN ASSIGN IR01.Cmd_Temp:=(9)
button at (120,230)-(201,251): text "23°C"; runs INTERN ASSIGN IR01.Cmd_Temp:=(10)
button at (120,260)-(201,281): text "24°C"; runs INTERN ASSIGN IR01.Cmd_Temp:=(11)
button at (120,350)-(201,371): text "27°C"; runs INTERN ASSIGN IR01.Cmd_Temp:=(14)
button at (120,320)-(201,341): text "26°C"; runs INTERN ASSIGN IR01.Cmd_Temp:=(13)
button at (120,290)-(201,311): text "25°C"; runs INTERN ASSIGN IR01.Cmd_Temp:=(12)
rectangle at (680,100)-(771,121): text "%d"; shows IR01.SetOnOff
rectangle at (680,160)-(771,181): text "%d"; shows (IR01.SetCmdMode)-18
rectangle at (680,190)-(771,211): text "%d"; shows (IR01.SetCmdFan)-14
rectangle at (680,220)-(771,241): text "%d"; shows (IR01.SetCmdSwing)-22
rectangle at (20,10)-(781,41): text "IR-712A"
button at (470,300)-(551,321): text "ZTHL01"
rectangle at (560,270)-(601,291): text "T [°C]"
rectangle at (600,270)-(641,291): text "RH [%]"
rectangle at (640,270)-(691,291): text "FLUX [lx]"
rectangle at (690,270)-(751,291): text "VBATT [V]"
rectangle at (750,270)-(791,291): text "LQI"
rectangle at (560,300)-(601,321): text "%1.1f"; shows WORD_TO_REAL(ZTHL01.OUT_TEMP)/10
rectangle at (600,300)-(641,321): text "%d"; shows ZTHL01.OUT_HYGRO
rectangle at (640,300)-(691,321): text "%d"; shows ZTHL01.OUT_LUX
rectangle at (690,300)-(751,321): text "%1.2f"; shows WORD_TO_REAL(ZTHL01.OUT_VBATT)/100
rectangle at (750,300)-(791,321): text "%d"; shows ZTHL01.OUT_LQI
button at (710,360)-(781,401): text "HOME"; opens PLC_Visu
6 more shapes without text or variables
9 elements of other kinds (tables, trends, ...) not read
*)

(* Visualisation PLC_VISU
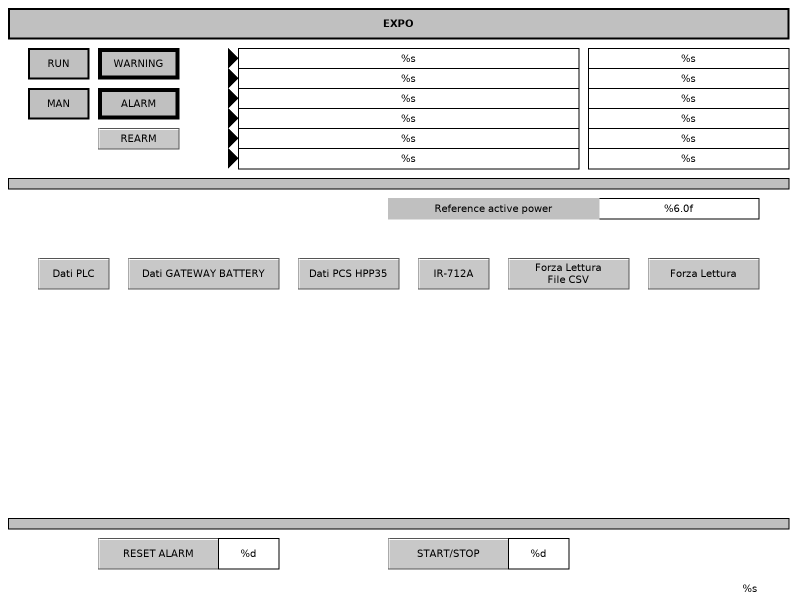
rectangle at (520,570)-(761,591): text "%s"; shows Sys.Time_LogString
rectangle at (10,0)-(791,31): text "EXPO"
rounded rectangle at (30,40)-(91,71): text "RUN"; alarm colour if NOT Mode_Manual; runs INTERN ASSIGN Mode_Manual:=(FALSE)
rounded rectangle at (30,80)-(91,111): text "MAN"; alarm colour if Mode_Manual; runs INTERN ASSIGN Mode_Manual:=(TRUE)
button at (40,250)-(111,281): text "Dati PLC"; opens WebVisu_PLC
rectangle at (590,40)-(791,61): text "%s"; shows Sys.LastLogs_Msg[0]
polygon at (230,140)-(240,160): invisible if Sys.LastLogs_Idx<>0
rectangle at (590,60)-(791,81): text "%s"; shows Sys.LastLogs_Msg[1]
polygon at (230,40)-(240,60): invisible if Sys.LastLogs_Idx<>1
rectangle at (590,80)-(791,101): text "%s"; shows Sys.LastLogs_Msg[2]
polygon at (230,60)-(240,80): invisible if Sys.LastLogs_Idx<>2
rectangle at (590,100)-(791,121): text "%s"; shows Sys.LastLogs_Msg[3]
polygon at (230,80)-(240,100): invisible if Sys.LastLogs_Idx<>3
rectangle at (590,120)-(791,141): text "%s"; shows Sys.LastLogs_Msg[4]
polygon at (230,100)-(240,120): invisible if Sys.LastLogs_Idx<>4
rectangle at (590,140)-(791,161): text "%s"; shows Sys.LastLogs_Msg[5]
polygon at (230,120)-(240,140): invisible if Sys.LastLogs_Idx<>5
rectangle at (240,40)-(581,61): text "%s"; shows Sys.LastLogs_Dat[0]
rectangle at (240,60)-(581,81): text "%s"; shows Sys.LastLogs_Dat[1]
rectangle at (240,80)-(581,101): text "%s"; shows Sys.LastLogs_Dat[2]
rectangle at (240,100)-(581,121): text "%s"; shows Sys.LastLogs_Dat[3]
rectangle at (240,120)-(581,141): text "%s"; shows Sys.LastLogs_Dat[4]
rectangle at (240,140)-(581,161): text "%s"; shows Sys.LastLogs_Dat[5]
rectangle at (100,80)-(181,111): text "ALARM"; alarm colour if Sys.Alarm; runs INTERN ASSIGN Mode_Manual:=(FALSE)
rectangle at (100,40)-(181,71): text "WARNING"; alarm colour if Sys.Warning; runs INTERN ASSIGN Mode_Manual:=(TRUE)
button at (100,120)-(181,141): text "REARM"; runs INTERN ASSIGN Sys.Alarm:=(FALSE);INTERN ASSIGN Sys.Warning:=(FALSE)
button at (650,250)-(761,281): text "Forza Lettura"; taps .ForzaLettura
rectangle at (600,190)-(761,211): text "%6.0f"; shows .Ref_P
rectangle at (390,190)-(601,211): text "Reference active power"
button at (130,250)-(281,281): text "Dati GATEWAY BATTERY"; opens WebVisu_GW
button at (300,250)-(401,281): text "Dati PCS HPP35"; opens WebVisu_PCS
button at (510,250)-(631,281): text "Forza Lettura / File CSV"; taps .ForzaLetturaCSV
button at (100,530)-(221,561): text "RESET ALARM"; runs INTERN ASSIGN wbResetAlarm:=(TRUE)
button at (390,530)-(511,561): text "START/STOP"; toggles wbStart_StopSystem; runs INTERN ASSIGN wbResetAlarm:=(TRUE)
rectangle at (220,530)-(281,561): text "%d"; shows wbResetAlarm
rectangle at (510,530)-(571,561): text "%d"; shows wbStart_StopSystem
button at (420,250)-(491,281): text "IR-712A"; opens IR_VISU
2 more shapes without text or variables
3 elements of other kinds (tables, trends, ...) not read
*)

(* Visualisation WEBVISU_GW
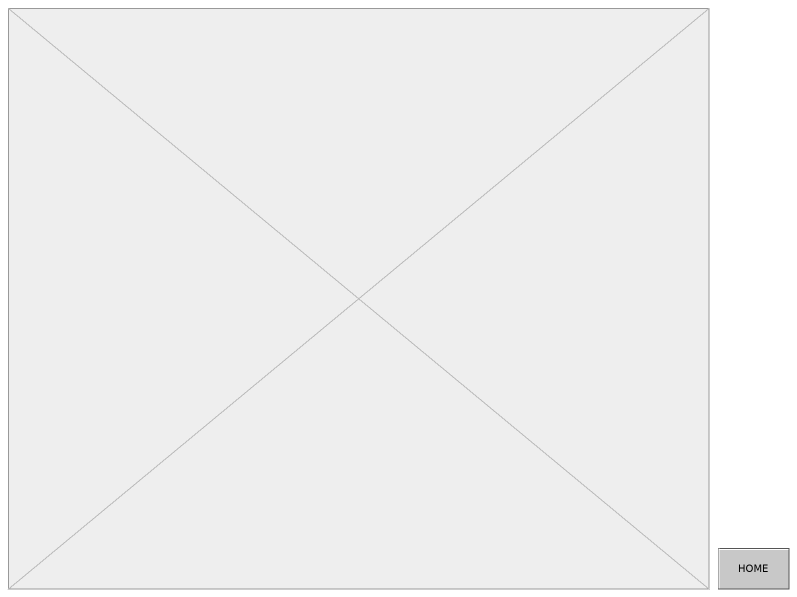
bitmap at (10,10)-(711,591): c:\users\esprinet 2014\documents\imi service\commesse\imi 15-438 expo\sviluppo\immagini\catturagw.jpg
button at (720,550)-(791,591): text "HOME"; opens PLC_Visu
26 elements of other kinds (tables, trends, ...) not read
*)

(* Visualisation WEBVISU_PCS
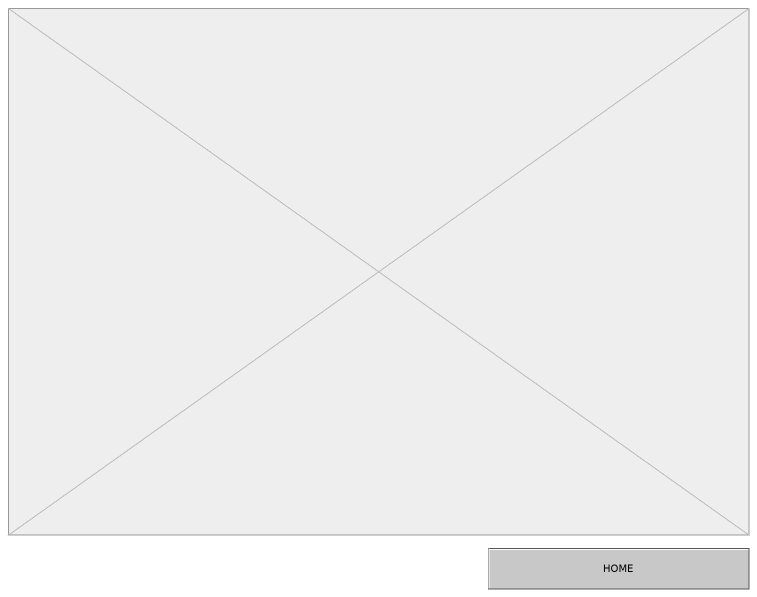
bitmap at (10,10)-(751,537): c:\users\esprinet 2014\documents\imi service\commesse\imi 15-438 expo\sviluppo\immagini\catturapcs.jpg
button at (490,550)-(751,591): text "HOME"; opens PLC_Visu
24 elements of other kinds (tables, trends, ...) not read
*)

(* Visualisation WEBVISU_PLC
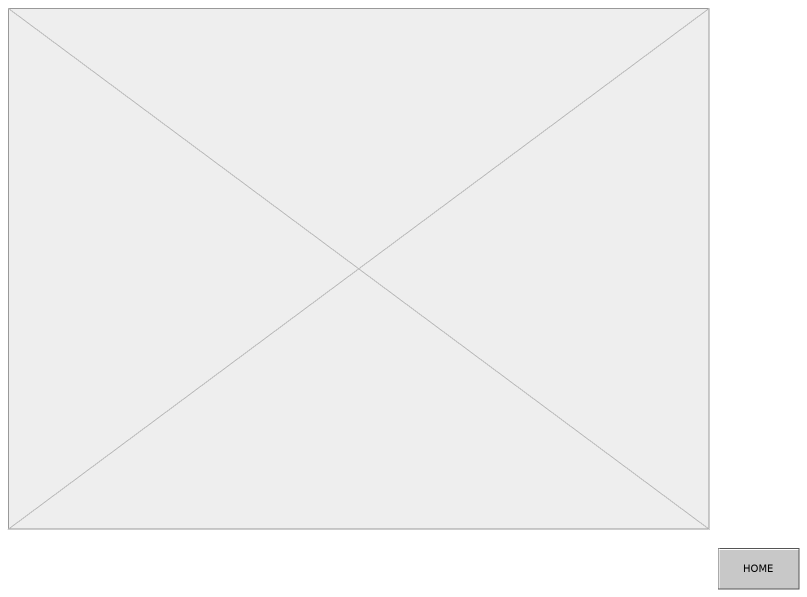
bitmap at (0,10)-(701,531): c:\users\esprinet 2014\documents\imi service\commesse\imi 15-438 expo\sviluppo\immagini\catturaplc.jpg
button at (710,550)-(791,591): text "HOME"; opens PLC_Visu
19 elements of other kinds (tables, trends, ...) not read
*)
